(* PLC project SafeLOGIC-1, BrAutomation SafeDESIGNER  4.4.0.0 *)
(* stored: companyURL http://www.br-automation.com, creationDateTime Mon May 10 15:18:37 2021 *)

PROGRAM Main
  VAR  (* added by the conversion: wires and edge detectors of the diagram *)
    _AND_S11_OUT : ANY;
    _SAFEBOOL_TO_BOOL67_OUT : BOOL;
  END_VAR

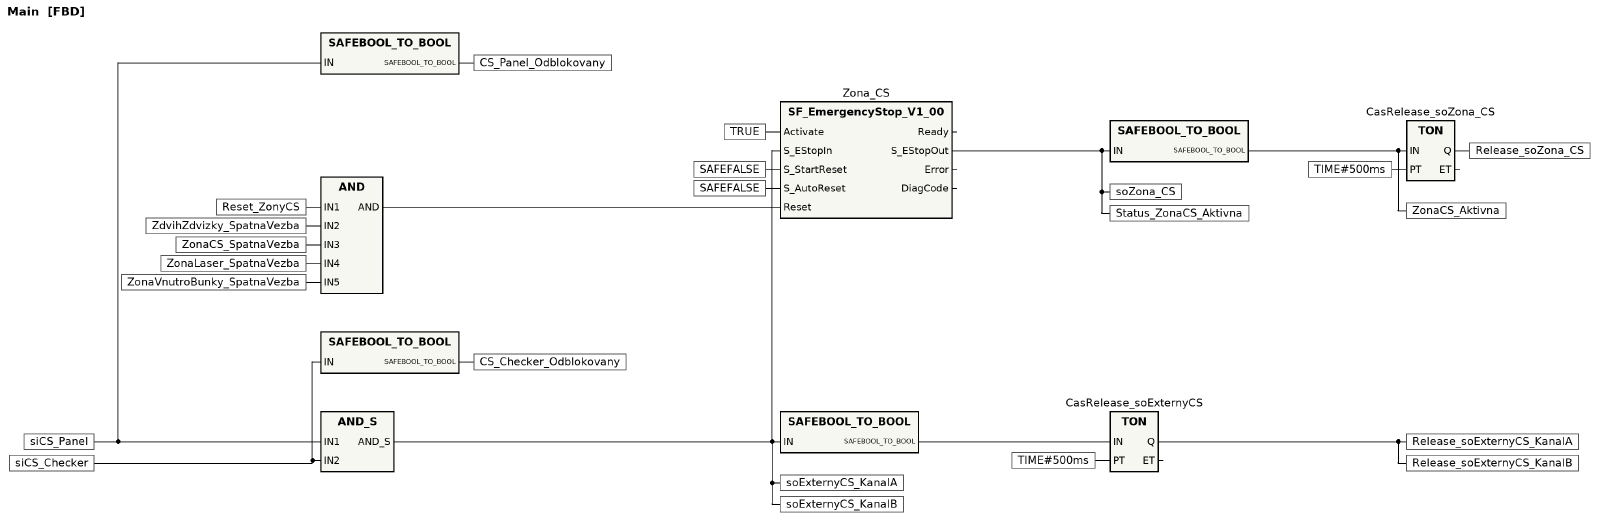
(* FBD diagram, written out as Structured Text *)
_AND_S11_OUT := AND_S(siCS_Panel, siCS_Checker);
Zona_CS(Activate := TRUE, S_EStopIn := _AND_S11_OUT, S_StartReset := SAFEFALSE, S_AutoReset := SAFEFALSE, Reset := Reset_ZonyCS AND ZdvihZdvizky_SpatnaVezba AND ZonaCS_SpatnaVezba AND ZonaLaser_SpatnaVezba AND ZonaVnutroBunky_SpatnaVezba);
soZona_CS := Zona_CS.S_EStopOut;
Status_ZonaCS_Aktivna := Zona_CS.S_EStopOut;
CS_Panel_Odblokovany := SAFEBOOL_TO_BOOL(siCS_Panel);
soExternyCS_KanalA := _AND_S11_OUT;
soExternyCS_KanalB := _AND_S11_OUT;
_SAFEBOOL_TO_BOOL67_OUT := SAFEBOOL_TO_BOOL(Zona_CS.S_EStopOut);
CasRelease_soZona_CS(IN := _SAFEBOOL_TO_BOOL67_OUT, PT := TIME#500ms);
Release_soZona_CS := CasRelease_soZona_CS.Q;
CasRelease_soExternyCS(IN := SAFEBOOL_TO_BOOL(_AND_S11_OUT), PT := TIME#500ms);
Release_soExternyCS_KanalB := CasRelease_soExternyCS.Q;
Release_soExternyCS_KanalA := CasRelease_soExternyCS.Q;
ZonaCS_Aktivna := _SAFEBOOL_TO_BOOL67_OUT;
CS_Checker_Odblokovany := SAFEBOOL_TO_BOOL(siCS_Checker);
END_PROGRAM
